# B&R Automation Studio project MirrElszkowskischody
Automation Studio 3.0.90.38 SP20; Default project

## Configuration 4PP481

### Task classes (Cpu.sw)
```
Cyclic#4:
  Zarowa <- Zarowa.prg
  schody <- schody.prg
  Ppoz <- Ppoz.prg
```

## Configuration Simulation

### Task classes (Cpu.sw)
```
Cyclic#4:
  Zarowa <- Zarowa.prg
  schody <- schody.prg
  Ppoz <- Ppoz.prg
Libraries: AsIecCon, astime
```

## Logical view

Binary libraries used (declarations not repeated): RUNTIME, Operator, AsIecCon, astime


### Program Logical/schody (IEC) - A new program

#### schody.var
```iecst
(********************************************************************
 * COPYRIGHT --
 ********************************************************************
 * Program: schody
 * File: schody.var
 * Author: User
 * Created: November 16, 2017
 ********************************************************************
 * Local variables of program schody
 ********************************************************************)
VAR
	doZarowka : ARRAY[0..9] OF BOOL;
	diPrzelacznik : ARRAY[0..9] OF BOOL;
	diCzujnikSwiatla : BOOL := FALSE;
END_VAR
```

#### schody.ab
```automation-basic
(********************************************************************
 * COPYRIGHT --
 ********************************************************************
 * Program: schody
 * File: schody.ab
 * Author: User
 * Created: November 16, 2017
 ********************************************************************
 * Implementation of program schody
 ********************************************************************)

PROGRAM _INIT

(* TODO : Add your code here *)

END_PROGRAM

PROGRAM _CYCLIC

doZarowka[0] = (diPrzelacznik[0] XOR diPrzelacznik[1]) AND diCzujnikSwiatla

END_PROGRAM

PROGRAM _EXIT

(* TODO : Add your code here *)

END_PROGRAM
```

### Program Logical/Ppoz (IEC) - A new program

#### Ppoz.ab - Implementation code
```automation-basic
(********************************************************************
 * COPYRIGHT --
 ********************************************************************
 * Program: Ppoz
 * File: Ppoz.ab
 * Author: User
 * Created: November 16, 2017
 ********************************************************************
 * Implementation of program Ppoz
 ********************************************************************)

PROGRAM _INIT

	uiModeWork = 2

END_PROGRAM

PROGRAM _CYCLIC
	CASE uiModeWork OF
		ACTION 1:
			Room[0].doTryskacz = Room[0].uiTryskacz
			System.doKogut = System.uiKogut
			System.doSyrena = System.uiSyrena
			ENDACTION
		ACTION 2:
			System.doSystemAktywny = ((System.diStart OR System.doSystemAktywny) AND NOT(System.diStop))
			IF System.doSystemAktywny THEN
				Room[0].doTryskacz = (Room[0].diCzujnikDym AND Room[0].diCzujnikSwiatlo AND NOT (Room[0].diCzujnikTemp)) OR  \
				(Room[0].diCzujnikDym AND NOT (Room[0].diCzujnikSwiatlo) AND Room[0].diCzujnikTemp) OR \
				(NOT (Room[0].diCzujnikDym) AND Room[0].diCzujnikSwiatlo AND Room[0].diCzujnikTemp) OR \
				(Room[0].diCzujnikDym AND Room[0].diCzujnikSwiatlo AND Room[0].diCzujnikTemp)
					System.doSyrena = Room[0].doTryskacz AND NOT(System.diReset)
					System.doKogut = Room[0].doTryskacz
				ELSE
					Room[0].doTryskacz = FALSE
					System.doSyrena = FALSE
					System.doKogut = FALSE

				ENDIF
		ENDACTION
ENDCASE
END_PROGRAM

PROGRAM _EXIT

(* TODO : Add your code here *)

END_PROGRAM
```

#### Ppoz.var - Local variables
```iecst
(********************************************************************
 * COPYRIGHT --
 ********************************************************************
 * Program: Ppoz
 * File: Ppoz.var
 * Author: User
 * Created: November 16, 2017
 ********************************************************************
 * Local variables of program Ppoz
 ********************************************************************)
VAR
	System : SystemStruct;
	Room : ARRAY[0..9] OF RoomStruct := [10(0)];
	uiModeWork : USINT := 0;
END_VAR
```

Listed in the project but not available here: Logical/Global.var, Logical/Zarowa, Logical/Ppoz/Ppoz.typ
